(* Logix 5000 project; controller cal1632 1756-L62 rev 16.20; software revision 16.05; part 35 of 61 *)
(* tags used below, declared in another part *)
   FAULT : BOOL;
   HMI : BOOL;
   p01_param_min_start_tension : REAL;
   p01_recipe_active : recipe;
   p01r02_plc_scan_time_in_sec : REAL;
   p01r09_pb_global_reset : BOOL;
   p01r09_request_line_jog : BOOL;
   p01r09_stretch_mode : BOOL;
   p01r12_master_ramped_speed : REAL;
   p01r13_line_running : BOOL;
   p01r13_line_slow_ramp : BOOL;
   p01r13_permissive_drives : BOOL;
   p01r13_state : DINT;
   p02_real_from_hmi : hmi_real;
   p20r15_loa_on : BOOL;
   p20r16_lob_on : BOOL;
   p22_ai_speed : REAL;
   p22_ai_ts1_lc : REAL;
   p22_ao_selected_speed : REAL;
   p22_ao_torque : REAL;
   p22_control_word : INT;
   p22_di_brake : BOOL;
   p22_di_jog : BOOL;
   p22_di_jog_fwd : BOOL;
   p22_di_jog_rev : BOOL;
   p22_di_run : BOOL;
   p22_di_therm : BOOL;
   p22_dint_to_hmi : DINT[16];
   p22_param_ts1_jog_speed : REAL;
   p22_status_word : INT;
   p22_ts1_acc_rate : REAL;
   p22_ts1_decel_rate : REAL;
   p22_ts1_vfd : ABB_PROTOCOL_VFD;
   p22r02_tension_dev_max : REAL;
   p22r02_tension_dev_min : REAL;
   p22r08 : routine;
   p22r08_timer_fault : TIMER[4];
   p22r08_timer_warning : TIMER[4];
   p22r09 : routine;
   p22r09_mode_jog : BOOL;
   p22r09_mode_run : BOOL;
   p22r09_mode_thread : BOOL;
   p22r09_pb_jog_fwd : BOOL;
   p22r09_pb_jog_rev : BOOL;
   p22r09_timer_fault : TIMER[4];
   p22r09_timer_warning : TIMER[4];
   p22r10 : routine;
   p22r10_calc_speed_offset : REAL;
   p22r10_param_psn_gain : REAL;
   p22r10_pid_out : REAL;
   p22r10_pid_psn : PID;
   p22r10_pid_psn_cv : REAL;
   p22r10_pid_psn_pv : REAL;
   p22r10_selected_torque : REAL;
   p22r10_speed_offset : REAL;
   p22r10_stretch : REAL;
   p22r10_timer_fault : TIMER[4];
   p22r10_timer_warning : TIMER[4];
   p22r11 : routine;
   p22r11_acc_decel_ramp : SYS_ACC_DEC_RAMP;
   p22r11_permissive_jog : BOOL;
   p22r11_request_jog_fwd : BOOL;
   p22r11_request_jog_rev : BOOL;
   p22r11_request_line_jog : BOOL;
   p22r11_request_line_run : BOOL;
   p22r11_request_start : BOOL;
   p22r11_request_tension : BOOL;
   p22r11_request_thread_fwd : BOOL;
   p22r11_request_thread_rev : BOOL;
   p22r11_selected_speed : REAL;
   p22r11_timer_fault : TIMER[10];
   p22r11_timer_warning : TIMER[5];
   p22r11_zero_speed : BOOL;
   p23r15_pid_tension_control : BOOL;
   p25r09_mode_thread : BOOL;
   p25r09_pb_jog_fwd : BOOL;
   p25r09_pb_jog_rev : BOOL;
(* P22_Tension_Stand_1, continued *)

ROUTINE R08_Warnings   (* ladder *)
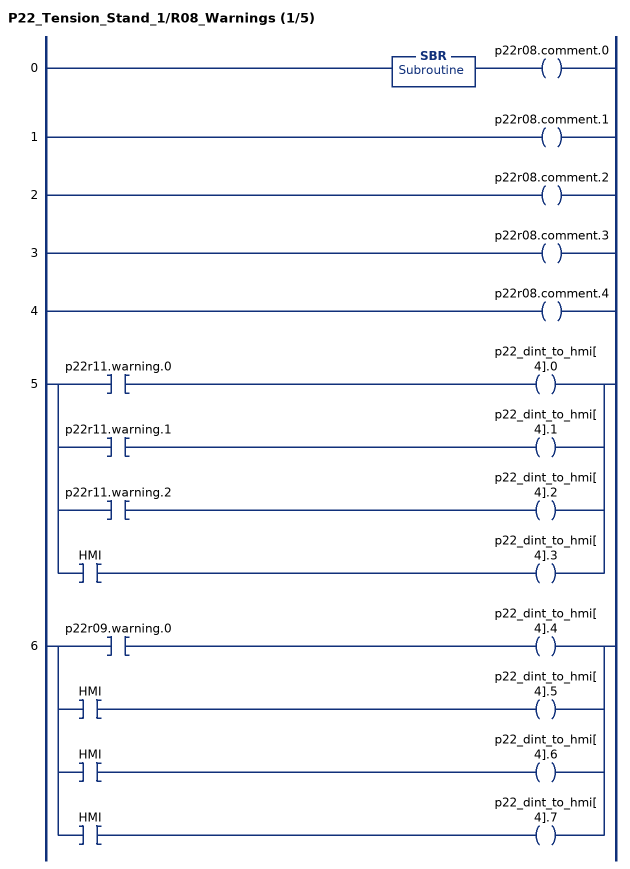
   0: SBR()OTE(p22r08.comment.0);
   1: OTE(p22r08.comment.1);
   2: OTE(p22r08.comment.2);
   3: OTE(p22r08.comment.3);
   4: OTE(p22r08.comment.4);
   5: [XIC(p22r11.warning.0) OTE(p22_dint_to_hmi[4].0) ,XIC(p22r11.warning.1) OTE(p22_dint_to_hmi[4].1) ,XIC(p22r11.warning.2) OTE(p22_dint_to_hmi[4].2) ,XIC(HMI) OTE(p22_dint_to_hmi[4].3) ];
   6: [XIC(p22r09.warning.0) OTE(p22_dint_to_hmi[4].4) ,XIC(HMI) OTE(p22_dint_to_hmi[4].5) ,XIC(HMI) OTE(p22_dint_to_hmi[4].6) ,XIC(HMI) OTE(p22_dint_to_hmi[4].7) ];
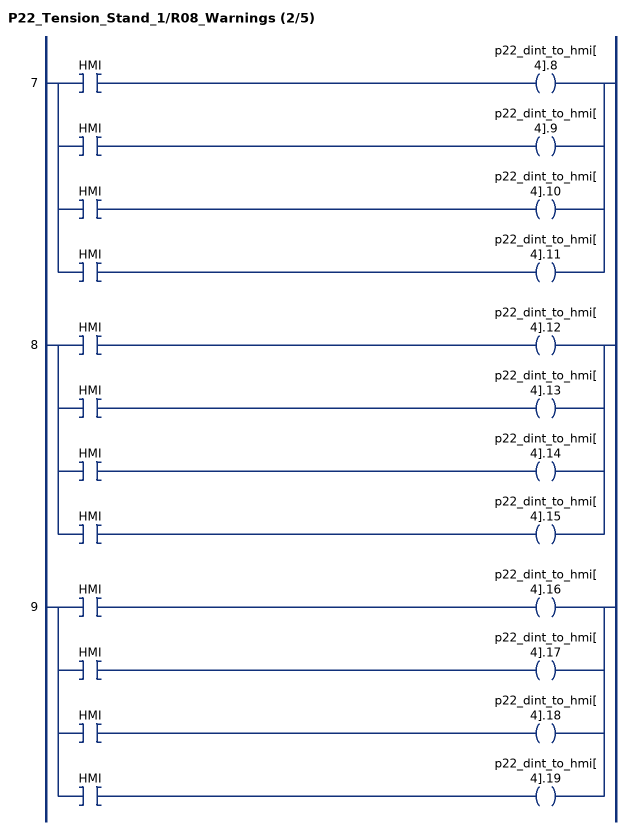
   7: [XIC(HMI) OTE(p22_dint_to_hmi[4].8) ,XIC(HMI) OTE(p22_dint_to_hmi[4].9) ,XIC(HMI) OTE(p22_dint_to_hmi[4].10) ,XIC(HMI) OTE(p22_dint_to_hmi[4].11) ];
   8: [XIC(HMI) OTE(p22_dint_to_hmi[4].12) ,XIC(HMI) OTE(p22_dint_to_hmi[4].13) ,XIC(HMI) OTE(p22_dint_to_hmi[4].14) ,XIC(HMI) OTE(p22_dint_to_hmi[4].15) ];
   9: [XIC(HMI) OTE(p22_dint_to_hmi[4].16) ,XIC(HMI) OTE(p22_dint_to_hmi[4].17) ,XIC(HMI) OTE(p22_dint_to_hmi[4].18) ,XIC(HMI) OTE(p22_dint_to_hmi[4].19) ];
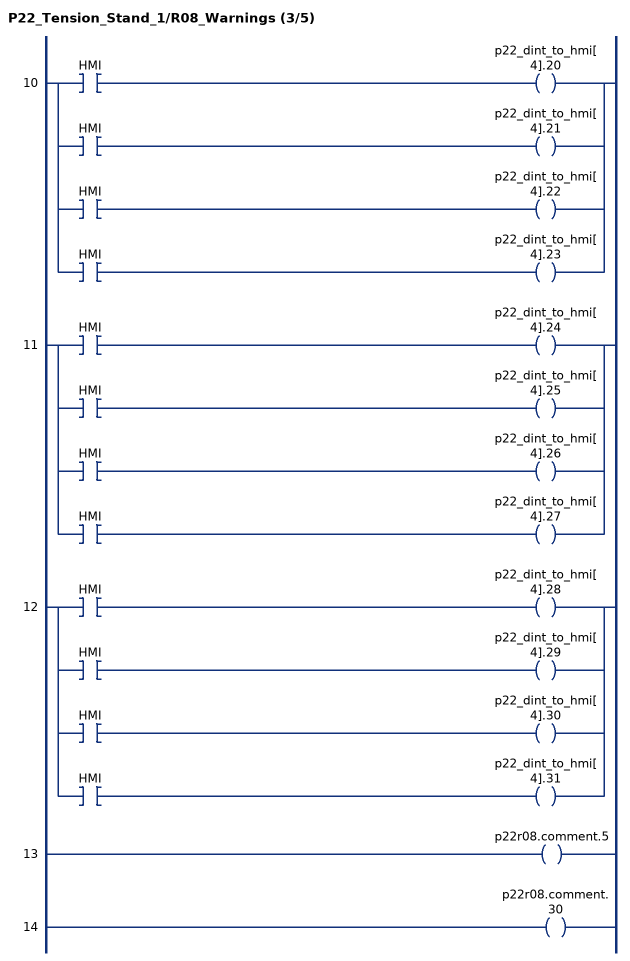
   10: [XIC(HMI) OTE(p22_dint_to_hmi[4].20) ,XIC(HMI) OTE(p22_dint_to_hmi[4].21) ,XIC(HMI) OTE(p22_dint_to_hmi[4].22) ,XIC(HMI) OTE(p22_dint_to_hmi[4].23) ];
   11: [XIC(HMI) OTE(p22_dint_to_hmi[4].24) ,XIC(HMI) OTE(p22_dint_to_hmi[4].25) ,XIC(HMI) OTE(p22_dint_to_hmi[4].26) ,XIC(HMI) OTE(p22_dint_to_hmi[4].27) ];
   12: [XIC(HMI) OTE(p22_dint_to_hmi[4].28) ,XIC(HMI) OTE(p22_dint_to_hmi[4].29) ,XIC(HMI) OTE(p22_dint_to_hmi[4].30) ,XIC(HMI) OTE(p22_dint_to_hmi[4].31) ];
   13: OTE(p22r08.comment.5);
   14: OTE(p22r08.comment.30);
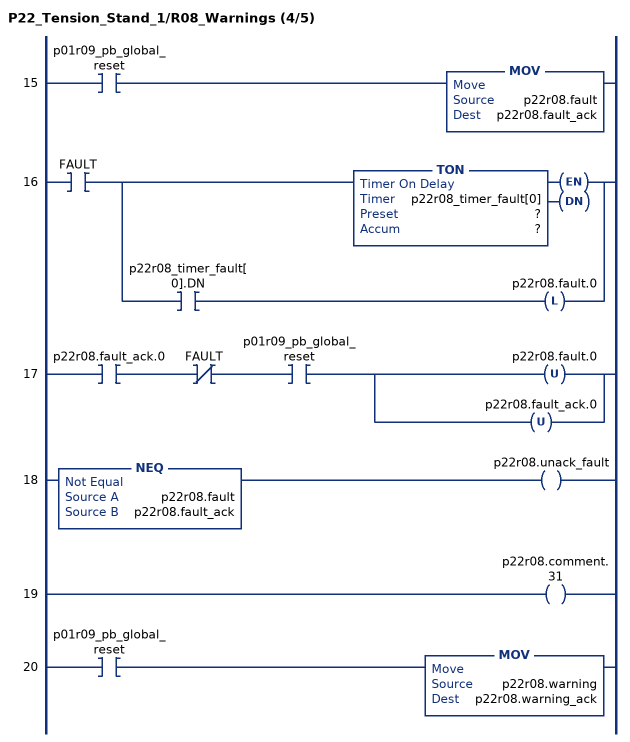
   15: XIC(p01r09_pb_global_reset)MOV(p22r08.fault,p22r08.fault_ack);
   16: XIC(FAULT)[TON(p22r08_timer_fault[0],?,?) ,XIC(p22r08_timer_fault[0].DN) OTL(p22r08.fault.0) ];
   17: XIC(p22r08.fault_ack.0)XIO(FAULT)XIC(p01r09_pb_global_reset)[OTU(p22r08.fault.0) ,OTU(p22r08.fault_ack.0) ];
   18: NEQ(p22r08.fault,p22r08.fault_ack)OTE(p22r08.unack_fault);
   19: OTE(p22r08.comment.31);
   20: XIC(p01r09_pb_global_reset)MOV(p22r08.warning,p22r08.warning_ack);
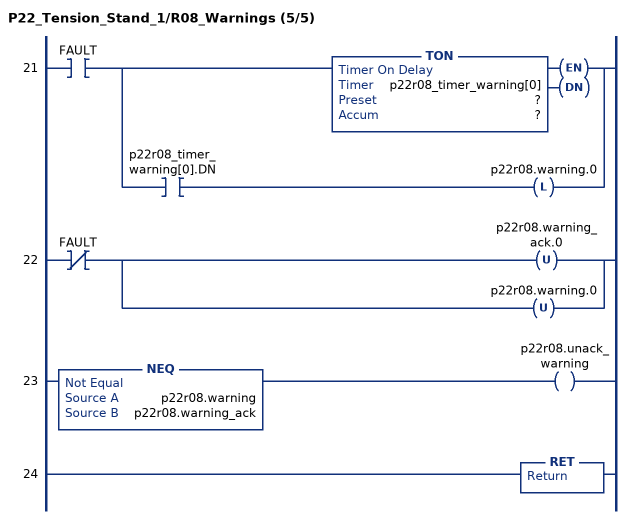
   21: XIC(FAULT)[TON(p22r08_timer_warning[0],?,?) ,XIC(p22r08_timer_warning[0].DN) OTL(p22r08.warning.0) ];
   22: XIO(FAULT)[OTU(p22r08.warning_ack.0) ,OTU(p22r08.warning.0) ];
   23: NEQ(p22r08.warning,p22r08.warning_ack)OTE(p22r08.unack_warning);
   24: RET();
END_ROUTINE

ROUTINE R09_Modes   (* ladder *)
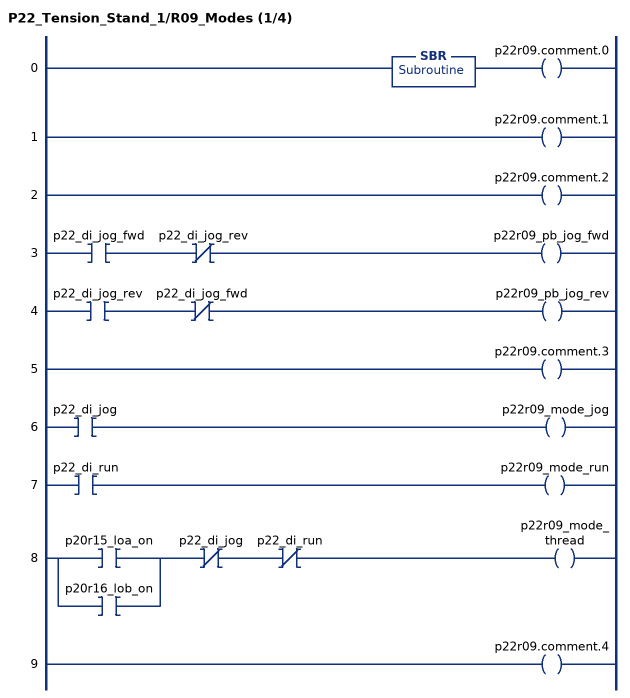
   0: SBR()OTE(p22r09.comment.0);
   1: OTE(p22r09.comment.1);
   2: OTE(p22r09.comment.2);
   3: XIC(p22_di_jog_fwd)XIO(p22_di_jog_rev)OTE(p22r09_pb_jog_fwd);
   4: XIC(p22_di_jog_rev)XIO(p22_di_jog_fwd)OTE(p22r09_pb_jog_rev);
   5: OTE(p22r09.comment.3);
   6: XIC(p22_di_jog)OTE(p22r09_mode_jog);
   7: XIC(p22_di_run)OTE(p22r09_mode_run);
   8: [XIC(p20r15_loa_on) ,XIC(p20r16_lob_on) ]XIO(p22_di_jog)XIO(p22_di_run)OTE(p22r09_mode_thread);
   9: OTE(p22r09.comment.4);
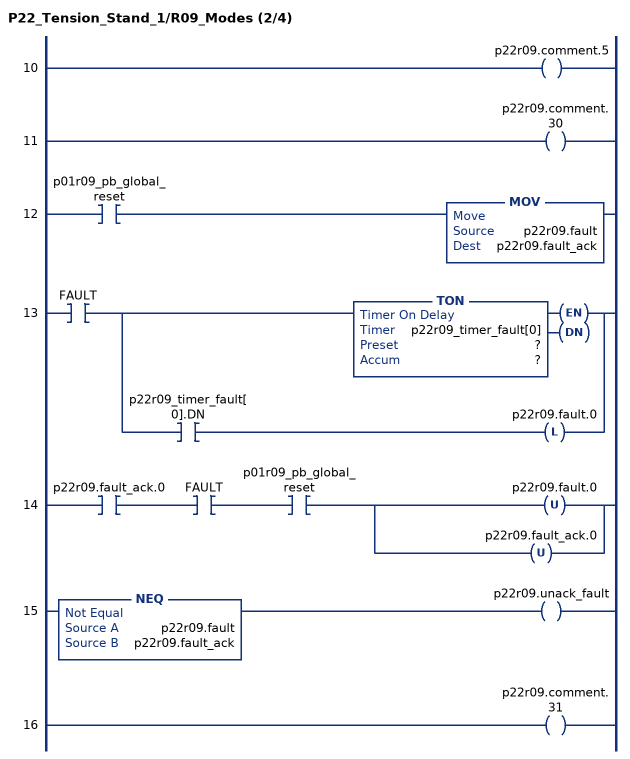
   10: OTE(p22r09.comment.5);
   11: OTE(p22r09.comment.30);
   12: XIC(p01r09_pb_global_reset)MOV(p22r09.fault,p22r09.fault_ack);
   13: XIC(FAULT)[TON(p22r09_timer_fault[0],?,?) ,XIC(p22r09_timer_fault[0].DN) OTL(p22r09.fault.0) ];
   14: XIC(p22r09.fault_ack.0)XIC(FAULT)XIC(p01r09_pb_global_reset)[OTU(p22r09.fault.0) ,OTU(p22r09.fault_ack.0) ];
   15: NEQ(p22r09.fault,p22r09.fault_ack)OTE(p22r09.unack_fault);
   16: OTE(p22r09.comment.31);
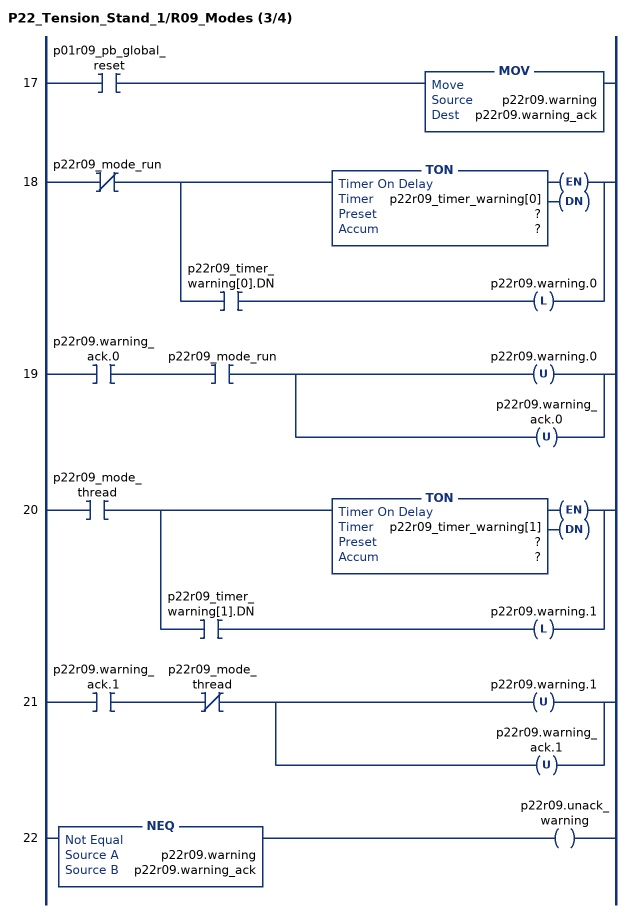
   17: XIC(p01r09_pb_global_reset)MOV(p22r09.warning,p22r09.warning_ack);
   18: XIO(p22r09_mode_run)[TON(p22r09_timer_warning[0],?,?) ,XIC(p22r09_timer_warning[0].DN) OTL(p22r09.warning.0) ];
   19: XIC(p22r09.warning_ack.0)XIC(p22r09_mode_run)[OTU(p22r09.warning.0) ,OTU(p22r09.warning_ack.0) ];
   20: XIC(p22r09_mode_thread)[TON(p22r09_timer_warning[1],?,?) ,XIC(p22r09_timer_warning[1].DN) OTL(p22r09.warning.1) ];
   21: XIC(p22r09.warning_ack.1)XIO(p22r09_mode_thread)[OTU(p22r09.warning.1) ,OTU(p22r09.warning_ack.1) ];
   22: NEQ(p22r09.warning,p22r09.warning_ack)OTE(p22r09.unack_warning);
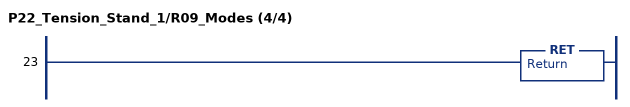
   23: RET();
END_ROUTINE

ROUTINE R10_Speed_Control   (* ladder *)
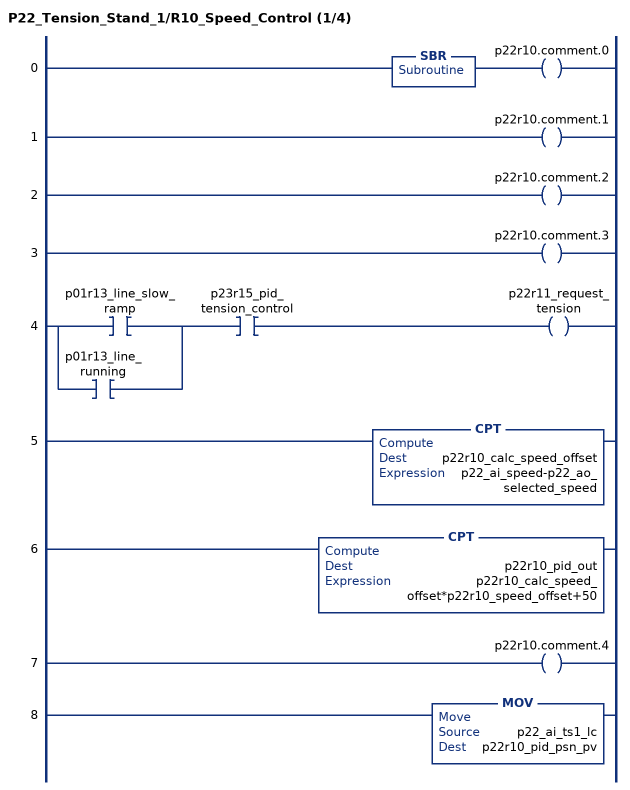
   0: SBR()OTE(p22r10.comment.0);
   1: OTE(p22r10.comment.1);
   2: OTE(p22r10.comment.2);
   3: OTE(p22r10.comment.3);
   4: [XIC(p01r13_line_slow_ramp) ,XIC(p01r13_line_running) ]XIC(p23r15_pid_tension_control)OTE(p22r11_request_tension);
   5: CPT(p22r10_calc_speed_offset,p22_ai_speed-p22_ao_selected_speed);
   6: CPT(p22r10_pid_out,p22r10_calc_speed_offset*p22r10_speed_offset+50);
   7: OTE(p22r10.comment.4);
   8: MOV(p22_ai_ts1_lc,p22r10_pid_psn_pv);
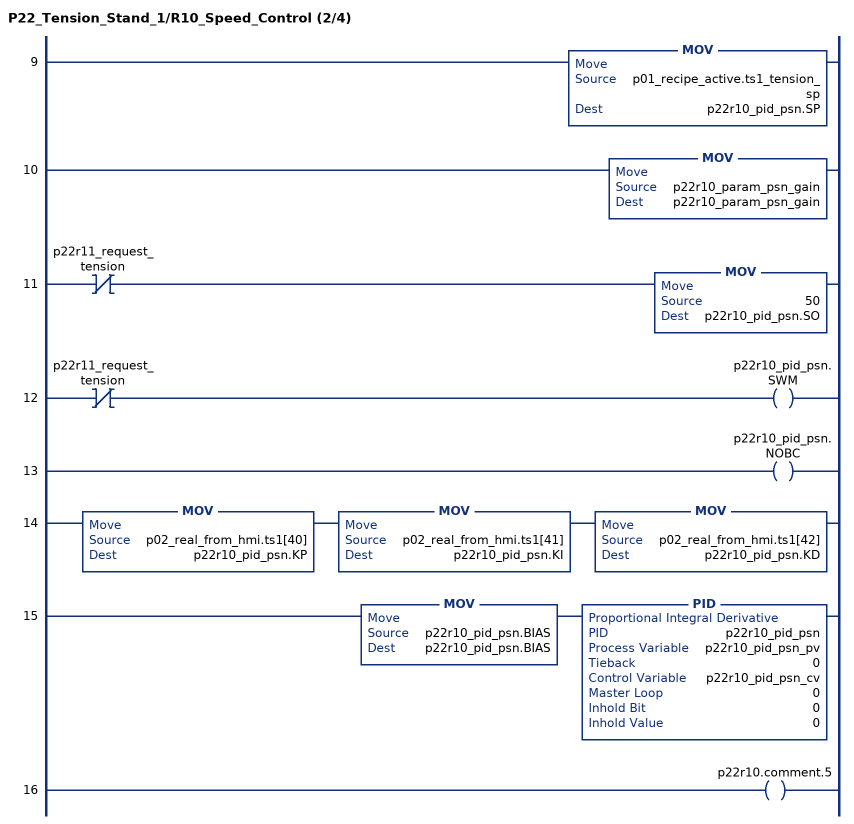
   9: MOV(p01_recipe_active.ts1_tension_sp,p22r10_pid_psn.SP);
   10: MOV(p22r10_param_psn_gain,p22r10_param_psn_gain);
   11: XIO(p22r11_request_tension)MOV(50,p22r10_pid_psn.SO);
   12: XIO(p22r11_request_tension)OTE(p22r10_pid_psn.SWM);
   13: OTE(p22r10_pid_psn.NOBC);
   14: MOV(p02_real_from_hmi.ts1[40],p22r10_pid_psn.KP)MOV(p02_real_from_hmi.ts1[41],p22r10_pid_psn.KI)MOV(p02_real_from_hmi.ts1[42],p22r10_pid_psn.KD);
   15: MOV(p22r10_pid_psn.BIAS,p22r10_pid_psn.BIAS)PID(p22r10_pid_psn,p22r10_pid_psn_pv,0,p22r10_pid_psn_cv,0,0,0);
   16: OTE(p22r10.comment.5);
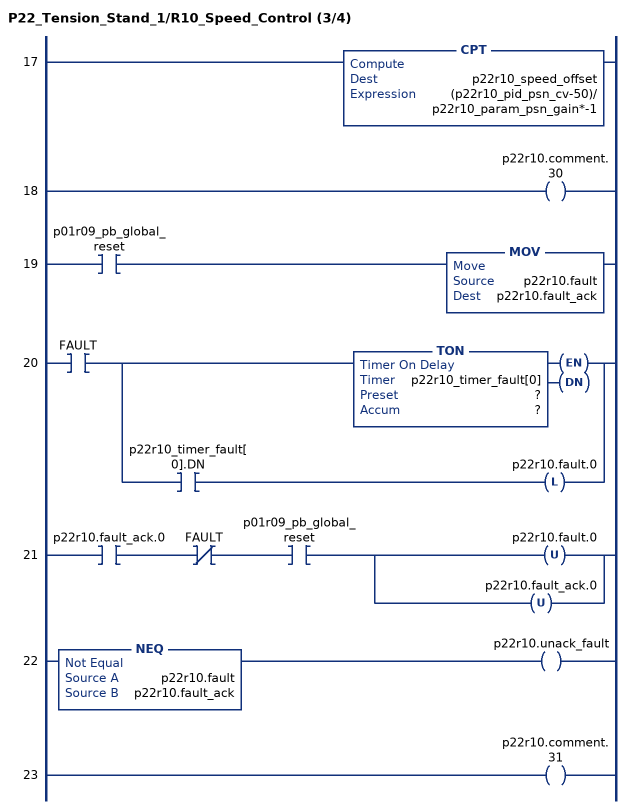
   17: CPT(p22r10_speed_offset,(p22r10_pid_psn_cv-50)/p22r10_param_psn_gain*-1);
   18: OTE(p22r10.comment.30);
   19: XIC(p01r09_pb_global_reset)MOV(p22r10.fault,p22r10.fault_ack);
   20: XIC(FAULT)[TON(p22r10_timer_fault[0],?,?) ,XIC(p22r10_timer_fault[0].DN) OTL(p22r10.fault.0) ];
   21: XIC(p22r10.fault_ack.0)XIO(FAULT)XIC(p01r09_pb_global_reset)[OTU(p22r10.fault.0) ,OTU(p22r10.fault_ack.0) ];
   22: NEQ(p22r10.fault,p22r10.fault_ack)OTE(p22r10.unack_fault);
   23: OTE(p22r10.comment.31);
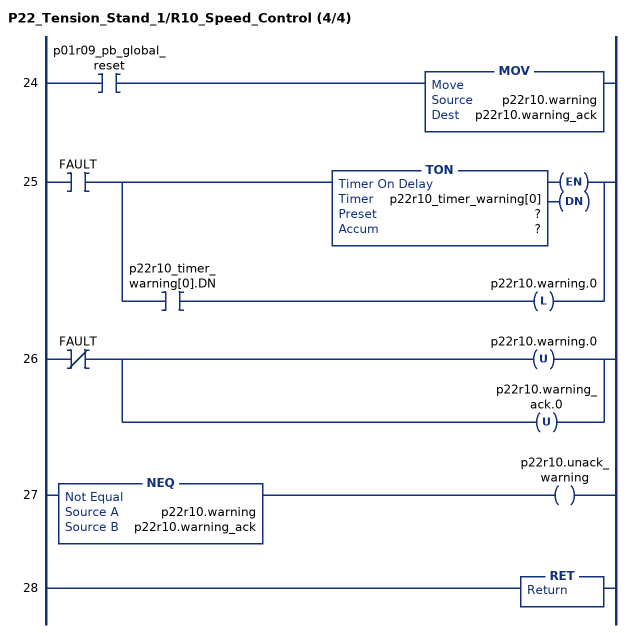
   24: XIC(p01r09_pb_global_reset)MOV(p22r10.warning,p22r10.warning_ack);
   25: XIC(FAULT)[TON(p22r10_timer_warning[0],?,?) ,XIC(p22r10_timer_warning[0].DN) OTL(p22r10.warning.0) ];
   26: XIO(FAULT)[OTU(p22r10.warning.0) ,OTU(p22r10.warning_ack.0) ];
   27: NEQ(p22r10.warning,p22r10.warning_ack)OTE(p22r10.unack_warning);
   28: RET();
END_ROUTINE

ROUTINE R11_VFD   (* ladder *)
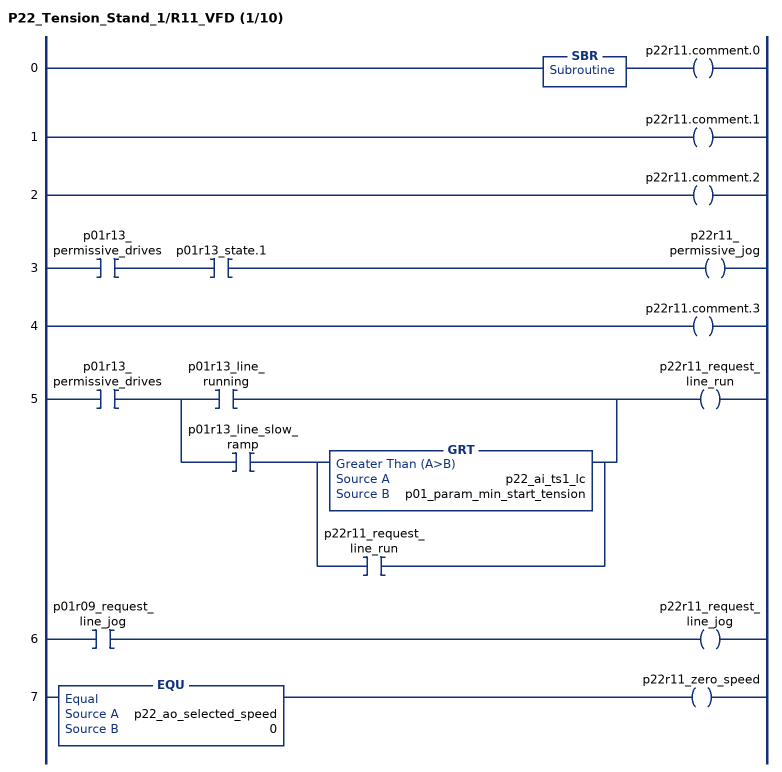
   0: SBR()OTE(p22r11.comment.0);
   1: OTE(p22r11.comment.1);
   2: OTE(p22r11.comment.2);
   3: XIC(p01r13_permissive_drives)XIC(p01r13_state.1)OTE(p22r11_permissive_jog);
   4: OTE(p22r11.comment.3);
   5: XIC(p01r13_permissive_drives)[XIC(p01r13_line_running) ,XIC(p01r13_line_slow_ramp) [GRT(p22_ai_ts1_lc,p01_param_min_start_tension) ,XIC(p22r11_request_line_run) ] ]OTE(p22r11_request_line_run);
   6: XIC(p01r09_request_line_jog)OTE(p22r11_request_line_jog);
   7: EQU(p22_ao_selected_speed,0)OTE(p22r11_zero_speed);
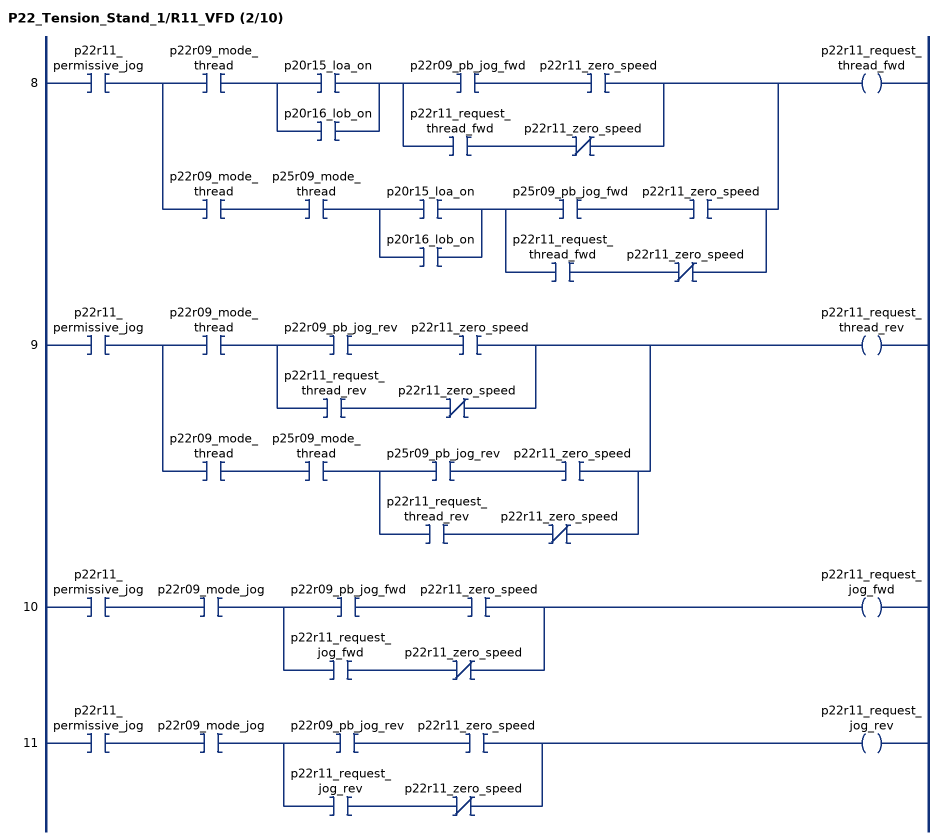
   8: XIC(p22r11_permissive_jog)[XIC(p22r09_mode_thread) [XIC(p20r15_loa_on) ,XIC(p20r16_lob_on) ] [XIC(p22r09_pb_jog_fwd) XIC(p22r11_zero_speed) ,XIC(p22r11_request_thread_fwd) XIO(p22r11_zero_speed) ] ,XIC(p22r09_mode_thread) XIC(p25r09_mode_thread) [XIC(p20r15_loa_on) ,XIC(p20r16_lob_on) ] [XIC(p25r09_pb_jog_fwd) XIC(p22r11_zero_speed) ,XIC(p22r11_request_thread_fwd) XIO(p22r11_zero_speed) ] ]OTE(p22r11_request_thread_fwd);
   9: XIC(p22r11_permissive_jog)[XIC(p22r09_mode_thread) [XIC(p22r09_pb_jog_rev) XIC(p22r11_zero_speed) ,XIC(p22r11_request_thread_rev) XIO(p22r11_zero_speed) ] ,XIC(p22r09_mode_thread) XIC(p25r09_mode_thread) [XIC(p25r09_pb_jog_rev) XIC(p22r11_zero_speed) ,XIC(p22r11_request_thread_rev) XIO(p22r11_zero_speed) ] ]OTE(p22r11_request_thread_rev);
   10: XIC(p22r11_permissive_jog)XIC(p22r09_mode_jog)[XIC(p22r09_pb_jog_fwd) XIC(p22r11_zero_speed) ,XIC(p22r11_request_jog_fwd) XIO(p22r11_zero_speed) ]OTE(p22r11_request_jog_fwd);
   11: XIC(p22r11_permissive_jog)XIC(p22r09_mode_jog)[XIC(p22r09_pb_jog_rev) XIC(p22r11_zero_speed) ,XIC(p22r11_request_jog_rev) XIO(p22r11_zero_speed) ]OTE(p22r11_request_jog_rev);
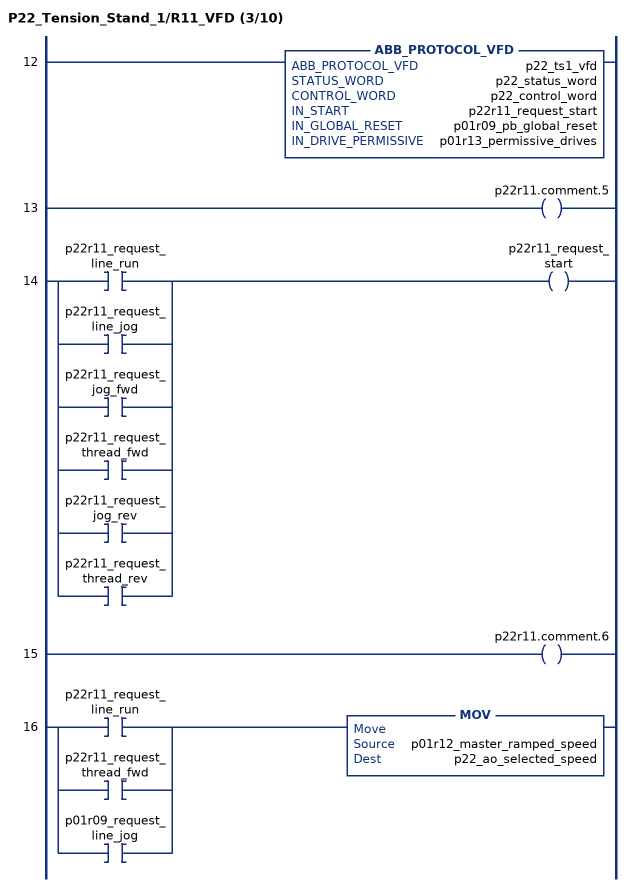
   12: ABB_PROTOCOL_VFD(p22_ts1_vfd,p22_status_word,p22_control_word,p22r11_request_start,p01r09_pb_global_reset,p01r13_permissive_drives);
   13: OTE(p22r11.comment.5);
   14: [XIC(p22r11_request_line_run) ,XIC(p22r11_request_line_jog) ,XIC(p22r11_request_jog_fwd) ,XIC(p22r11_request_thread_fwd) ,XIC(p22r11_request_jog_rev) ,XIC(p22r11_request_thread_rev) ]OTE(p22r11_request_start);
   15: OTE(p22r11.comment.6);
   16: [XIC(p22r11_request_line_run) ,XIC(p22r11_request_thread_fwd) ,XIC(p01r09_request_line_jog) ]MOV(p01r12_master_ramped_speed,p22_ao_selected_speed);
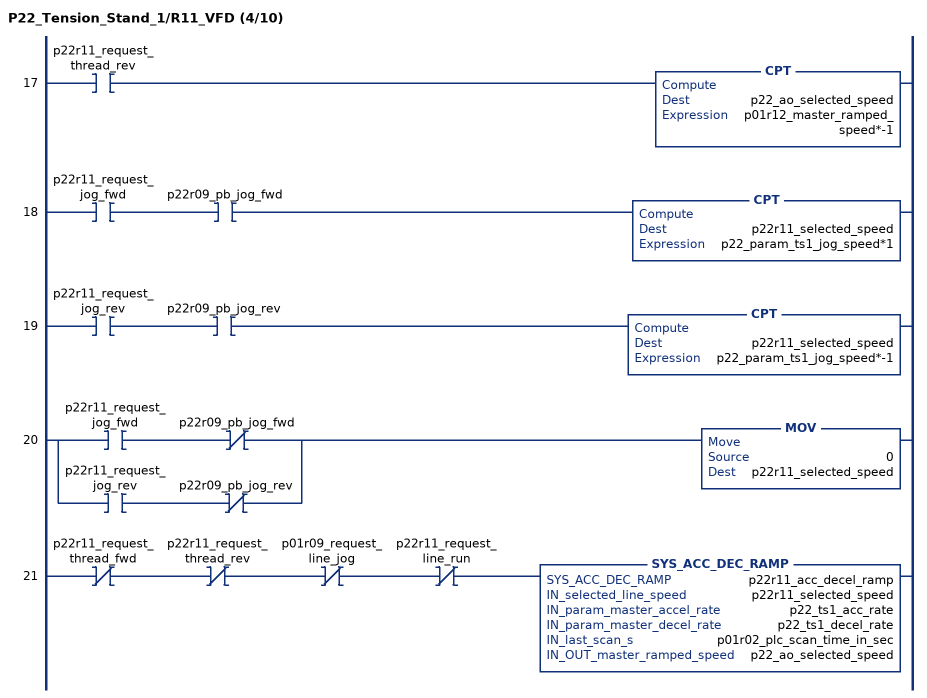
   17: XIC(p22r11_request_thread_rev)CPT(p22_ao_selected_speed,p01r12_master_ramped_speed*-1);
   18: XIC(p22r11_request_jog_fwd)XIC(p22r09_pb_jog_fwd)CPT(p22r11_selected_speed,p22_param_ts1_jog_speed*1);
   19: XIC(p22r11_request_jog_rev)XIC(p22r09_pb_jog_rev)CPT(p22r11_selected_speed,p22_param_ts1_jog_speed*-1);
   20: [XIC(p22r11_request_jog_fwd) XIO(p22r09_pb_jog_fwd) ,XIC(p22r11_request_jog_rev) XIO(p22r09_pb_jog_rev) ]MOV(0,p22r11_selected_speed);
   21: XIO(p22r11_request_thread_fwd)XIO(p22r11_request_thread_rev)XIO(p01r09_request_line_jog)XIO(p22r11_request_line_run)SYS_ACC_DEC_RAMP(p22r11_acc_decel_ramp,p22r11_selected_speed,p22_ts1_acc_rate,p22_ts1_decel_rate,p01r02_plc_scan_time_in_sec,p22_ao_selected_speed);
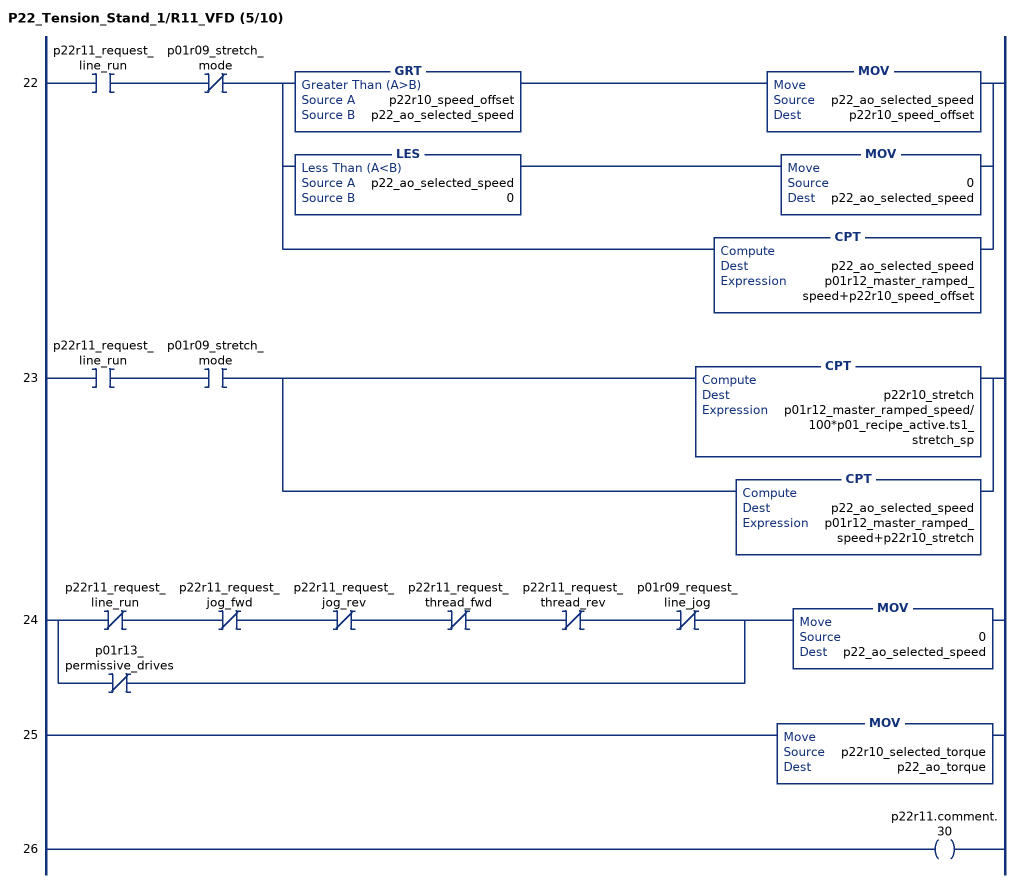
   22: XIC(p22r11_request_line_run)XIO(p01r09_stretch_mode)[GRT(p22r10_speed_offset,p22_ao_selected_speed) MOV(p22_ao_selected_speed,p22r10_speed_offset) ,LES(p22_ao_selected_speed,0) MOV(0,p22_ao_selected_speed) ,CPT(p22_ao_selected_speed,p01r12_master_ramped_speed+p22r10_speed_offset) ];
   23: XIC(p22r11_request_line_run)XIC(p01r09_stretch_mode)[CPT(p22r10_stretch,p01r12_master_ramped_speed/100*p01_recipe_active.ts1_stretch_sp) ,CPT(p22_ao_selected_speed,p01r12_master_ramped_speed+p22r10_stretch) ];
   24: [XIO(p22r11_request_line_run) XIO(p22r11_request_jog_fwd) XIO(p22r11_request_jog_rev) XIO(p22r11_request_thread_fwd) XIO(p22r11_request_thread_rev) XIO(p01r09_request_line_jog) ,XIO(p01r13_permissive_drives) ]MOV(0,p22_ao_selected_speed);
   25: MOV(p22r10_selected_torque,p22_ao_torque);
   26: OTE(p22r11.comment.30);
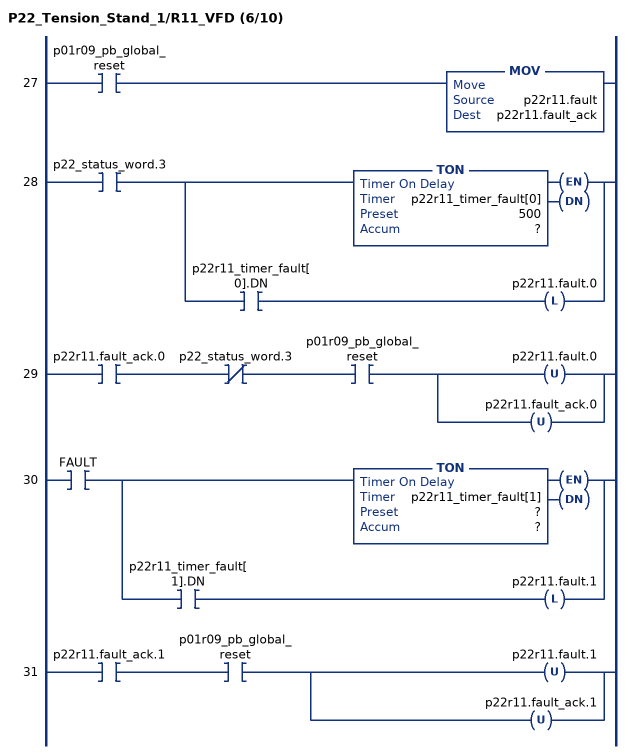
   27: XIC(p01r09_pb_global_reset)MOV(p22r11.fault,p22r11.fault_ack);
   28: XIC(p22_status_word.3)[TON(p22r11_timer_fault[0],?,?) ,XIC(p22r11_timer_fault[0].DN) OTL(p22r11.fault.0) ];
   29: XIC(p22r11.fault_ack.0)XIO(p22_status_word.3)XIC(p01r09_pb_global_reset)[OTU(p22r11.fault.0) ,OTU(p22r11.fault_ack.0) ];
   30: XIC(FAULT)[TON(p22r11_timer_fault[1],?,?) ,XIC(p22r11_timer_fault[1].DN) OTL(p22r11.fault.1) ];
   31: XIC(p22r11.fault_ack.1)XIC(p01r09_pb_global_reset)[OTU(p22r11.fault.1) ,OTU(p22r11.fault_ack.1) ];
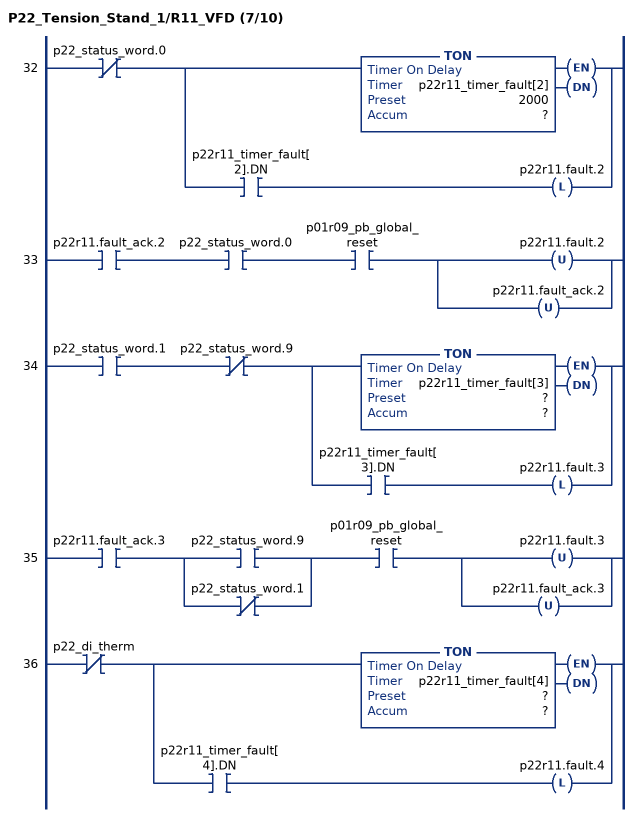
   32: XIO(p22_status_word.0)[TON(p22r11_timer_fault[2],?,?) ,XIC(p22r11_timer_fault[2].DN) OTL(p22r11.fault.2) ];
   33: XIC(p22r11.fault_ack.2)XIC(p22_status_word.0)XIC(p01r09_pb_global_reset)[OTU(p22r11.fault.2) ,OTU(p22r11.fault_ack.2) ];
   34: XIC(p22_status_word.1)XIO(p22_status_word.9)[TON(p22r11_timer_fault[3],?,?) ,XIC(p22r11_timer_fault[3].DN) OTL(p22r11.fault.3) ];
   35: XIC(p22r11.fault_ack.3)[XIC(p22_status_word.9) ,XIO(p22_status_word.1) ]XIC(p01r09_pb_global_reset)[OTU(p22r11.fault.3) ,OTU(p22r11.fault_ack.3) ];
   36: XIO(p22_di_therm)[TON(p22r11_timer_fault[4],?,?) ,XIC(p22r11_timer_fault[4].DN) OTL(p22r11.fault.4) ];
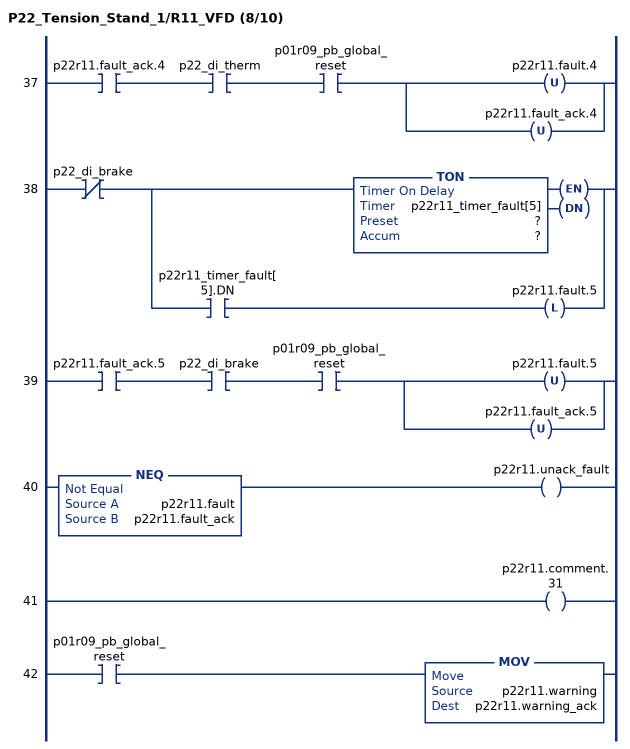
   37: XIC(p22r11.fault_ack.4)XIC(p22_di_therm)XIC(p01r09_pb_global_reset)[OTU(p22r11.fault.4) ,OTU(p22r11.fault_ack.4) ];
   38: XIO(p22_di_brake)[TON(p22r11_timer_fault[5],?,?) ,XIC(p22r11_timer_fault[5].DN) OTL(p22r11.fault.5) ];
   39: XIC(p22r11.fault_ack.5)XIC(p22_di_brake)XIC(p01r09_pb_global_reset)[OTU(p22r11.fault.5) ,OTU(p22r11.fault_ack.5) ];
   40: NEQ(p22r11.fault,p22r11.fault_ack)OTE(p22r11.unack_fault);
   41: OTE(p22r11.comment.31);
   42: XIC(p01r09_pb_global_reset)MOV(p22r11.warning,p22r11.warning_ack);
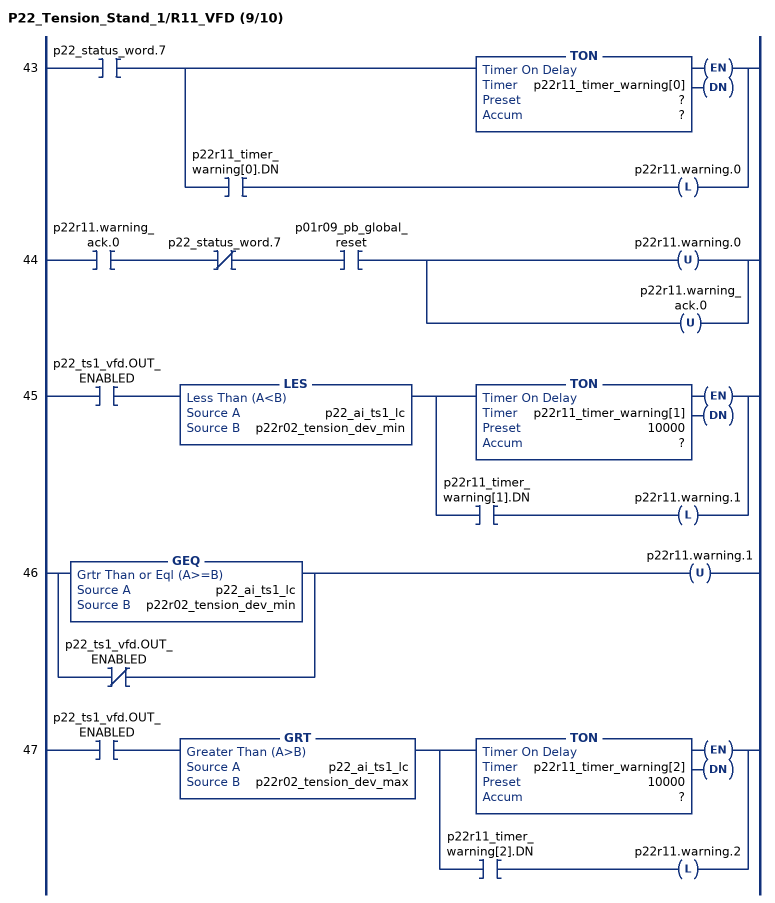
   43: XIC(p22_status_word.7)[TON(p22r11_timer_warning[0],?,?) ,XIC(p22r11_timer_warning[0].DN) OTL(p22r11.warning.0) ];
   44: XIC(p22r11.warning_ack.0)XIO(p22_status_word.7)XIC(p01r09_pb_global_reset)[OTU(p22r11.warning.0) ,OTU(p22r11.warning_ack.0) ];
   45: XIC(p22_ts1_vfd.OUT_ENABLED)LES(p22_ai_ts1_lc,p22r02_tension_dev_min)[TON(p22r11_timer_warning[1],?,?) ,XIC(p22r11_timer_warning[1].DN) OTL(p22r11.warning.1) ];
   46: [GEQ(p22_ai_ts1_lc,p22r02_tension_dev_min) ,XIO(p22_ts1_vfd.OUT_ENABLED) ]OTU(p22r11.warning.1);
   47: XIC(p22_ts1_vfd.OUT_ENABLED)GRT(p22_ai_ts1_lc,p22r02_tension_dev_max)[TON(p22r11_timer_warning[2],?,?) ,XIC(p22r11_timer_warning[2].DN) OTL(p22r11.warning.2) ];
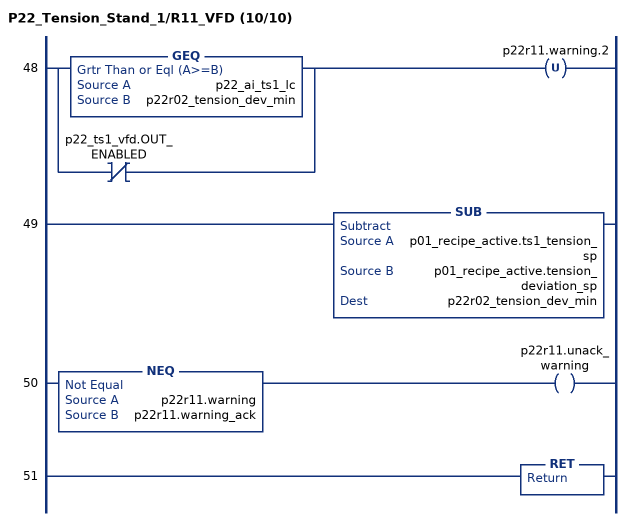
   48: [GEQ(p22_ai_ts1_lc,p22r02_tension_dev_min) ,XIO(p22_ts1_vfd.OUT_ENABLED) ]OTU(p22r11.warning.2);
   49: SUB(p01_recipe_active.ts1_tension_sp,p01_recipe_active.tension_deviation_sp,p22r02_tension_dev_min);
   50: NEQ(p22r11.warning,p22r11.warning_ack)OTE(p22r11.unack_warning);
   51: RET();
END_ROUTINE
END_PROGRAM
